(*
SPDX-FileCopyrightText: © 2026 Oleksandr Tiutyk <trofimich@gmail.com>
SPDX-License-Identifier: MIT
License: https://opensource.org/license/mit
*)

{attribute 'no_explicit_call' := 'do not call this function block directly'} 
{attribute 'enable_dynamic_creation'}
FUNCTION_BLOCK ABSTRACT CompositeCondition EXTENDS Condition IMPLEMENTS ICompositeCondition
VAR
	{attribute 'OPC.UA.DA' := '0'}
	_ClassName : STRING := __POUNAME();

	{attribute 'OPC.UA.DA' := '0'}
	_LogicalOperator : LOGICAL_OPERATOR;

	{attribute 'OPC.UA.DA' := '0'}
	_Children : TOF_Collections.List<0>(0);
END_VAR

METHOD AddChildCondition
VAR_INPUT
	condition : ICondition;
END_VAR
VAR
	argumentNullExcxeption : TOF_Core.ArgumentNotSpecifiedException;
END_VAR
IF condition = 0  THEN
	argumentNullExcxeption.Throw(NamespaceName, ClassName, __POUNAME(), __POSITION(), 'condition');
END_IF

condition.ParentCondition := THIS^;

_Children.AppendGeneric(TOF_Core.GenericValueFactory.FromParts(TOF_Core.GENERIC_TYPE_CLASS.OBJECT, condition.SelfAddress, condition.SelfSize, TOF_Core.GENERIC_MEMORY_MANAGEMENT_BEHAVIOR.STORE_ORIGINAL_REFERENCE_AND_NOT_OWNS_MEMORY));
END_METHOD

{attribute 'monitoring' := 'call'}
PROPERTY ClassName : REFERENCE TO STRING
GET
ClassName REF= _ClassName;
END_GET
END_PROPERTY

{attribute 'monitoring' := 'call'}
PROPERTY Configured : BOOL
GET
Configured := _Children.Length > 0;
END_GET
END_PROPERTY

PROPERTY LogicalOperator : LOGICAL_OPERATOR
GET
LogicalOperator := _LogicalOperator;
END_GET
SET
_LogicalOperator := LogicalOperator;
END_SET
END_PROPERTY

{attribute 'monitoring' := 'call'}
PROPERTY NamespaceName : REFERENCE TO STRING
GET
NamespaceName REF= CurrentNamespace.Name;
END_GET
END_PROPERTY

METHOD PROTECTED OnEvalute : BOOL
VAR_INPUT
	activity : IActivity;
END_VAR
VAR
	conditionException : TOF_Core.StandardException;

	i : DINT;
	
	childCondition : ICondition;
END_VAR
IF NOT Configured THEN
	conditionException.Throw(NamespaceName, ClassName, __POUNAME(), __POSITION(), TOF_Core.WideStrings.Concat255("Condition '", Name, "' is not configured"));
END_IF

IF _LogicalOperator = LOGICAL_OPERATOR.AND_ THEN
	OnEvalute := TRUE;	
END_IF
 
FOR i := 0 TO _Children.Length - 1 DO
	IF NOT __QUERYINTERFACE(_Children.Get(i).AsObject(), childCondition) THEN
		conditionException.Throw(NamespaceName, ClassName, __POUNAME(), __POSITION(), TOF_Core.WideStrings.Concat255("Condition #", TO_WSTRING(i), " is null"));
	END_IF
	
	IF NOT childCondition.Configured THEN
		conditionException.Throw(NamespaceName, ClassName, __POUNAME(), __POSITION(), TOF_Core.WideStrings.Concat255("Condition '", childCondition.Name, "' is not configured"));
	END_IF

	IF childCondition.Evaluate(activity) THEN
		IF _LogicalOperator = LOGICAL_OPERATOR.OR_ THEN
			OnEvalute := TRUE;	
			RETURN;
		END_IF
	ELSE
		IF _LogicalOperator = LOGICAL_OPERATOR.AND_ THEN
			OnEvalute := FALSE;	
			RETURN;
		END_IF
	END_IF	 
END_FOR
END_METHOD

{attribute 'monitoring' := 'call'}
PROPERTY SelfSize : ULINT
GET
SelfSize := XSIZEOF(THIS^);
END_GET
END_PROPERTY

END_FUNCTION_BLOCK

(* stored: Version 1.1.0.1
   POU CompositeCondition: Id {8a55c5b1-693f-4932-9f9a-010c3c539516}, SpecialFunc None
   Folder Overriden members: Id {92167edf-a171-45ae-b0b4-cbb4363d35a0}
   Method AddChildCondition: Id {a9ba8ac8-dab1-4579-a8c6-f1dcf4f0781e}
   Property ClassName: Id {70333ea1-3549-4d0a-a3ad-521d1db0db74}
   Get Get: Id {a5ccd782-e1de-457e-9e73-065fb67a7a80}
   Property Configured: Id {21dacc3f-ed62-4ab7-8da9-cb67ea9bfcba}
   Get Get: Id {ea5c9fa4-9f95-445e-834b-d8986cf079b5}
   Property LogicalOperator: Id {2e60dc3a-8843-4578-a90f-416536b1cdcb}
   Get Get: Id {24be606b-b29e-4d7a-9059-3d33397fc9bc}
   Set Set: Id {91bb16fb-1705-4e7d-aeac-ee32b7347b30}
   Property NamespaceName: Id {52983f0a-5112-4343-a340-1487d5e77845}
   Get Get: Id {8a11a0fb-561b-4d9a-b1ae-2ae3af60f58b}
   Method OnEvalute: Id {65421d01-d63f-414e-ae6f-3caad321436b}
   Property SelfSize: Id {0c774fc8-e3e1-46bd-bc7e-7d6910760a9c}
   Get Get: Id {02bdd4c2-e6e9-4e38-a963-e1672ee8a20b} *)
